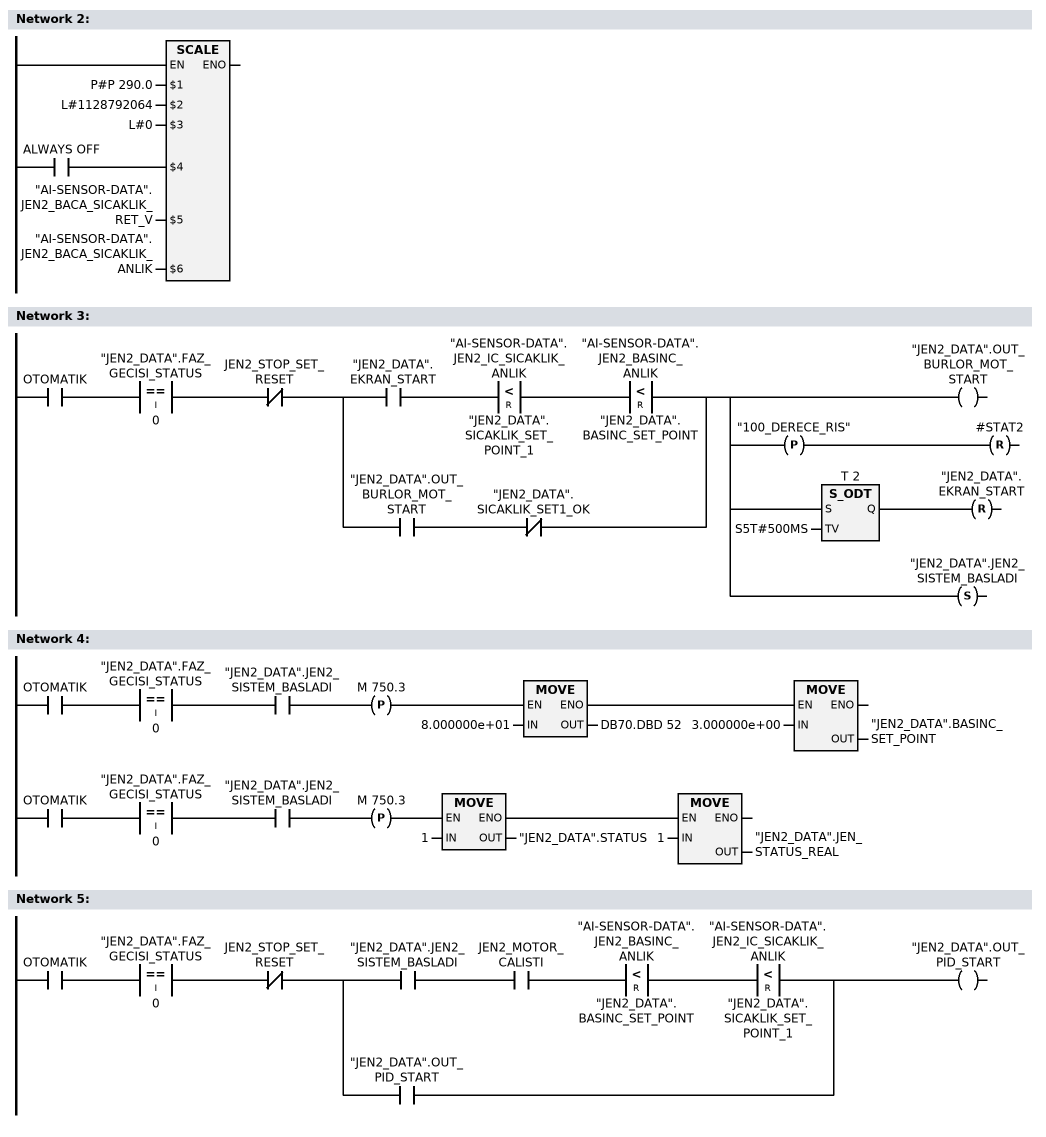
NETWORK
TITLE =
      A     "ALWAYS OFF";
      =     L 0.0;
      BLD   103;
      CALL  "SCALE" (
           $1                       := P#P 290.0,
           $2                       := L#1128792064,
           $3                       := L#0,
           $4                       := L 0.0,
           $5                       := "AI-SENSOR-DATA".JEN2_BACA_SICAKLIK_RET_V,
           $6                       := "AI-SENSOR-DATA".JEN2_BACA_SICAKLIK_ANLIK);
      NOP   0;
NETWORK
TITLE =
      A     "OTOMATIK";
      A(;
      L     "JEN2_DATA".FAZ_GECISI_STATUS;
      L     0;
      ==I;
      );
      AN    "JEN2_STOP_SET_RESET";
      A(;
      A     "JEN2_DATA".EKRAN_START;
      A(;
      L     "AI-SENSOR-DATA".JEN2_IC_SICAKLIK_ANLIK;
      L     "JEN2_DATA".SICAKLIK_SET_POINT_1;
      <R;
      );
      A(;
      L     "AI-SENSOR-DATA".JEN2_BASINC_ANLIK;
      L     "JEN2_DATA".BASINC_SET_POINT;
      <R;
      );
      O;
      A     "JEN2_DATA".OUT_BURLOR_MOT_START;
      AN    "JEN2_DATA".SICAKLIK_SET1_OK;
      );
      =     L 0.0;
      A     L 0.0;
      BLD   102;
      =     "JEN2_DATA".OUT_BURLOR_MOT_START;
      A     L 0.0;
      FP    "100_DERECE_RIS";
      R     #STAT2;
      A     L 0.0;
      L     S5T#500MS;
      SD    T 2;
      NOP   0;
      NOP   0;
      NOP   0;
      A     T 2;
      R     "JEN2_DATA".EKRAN_START;
      A     L 0.0;
      BLD   102;
      S     "JEN2_DATA".JEN2_SISTEM_BASLADI;
NETWORK
TITLE =
      A     "OTOMATIK";
      A(;
      L     "JEN2_DATA".FAZ_GECISI_STATUS;
      L     0;
      ==I;
      );
      A     "JEN2_DATA".JEN2_SISTEM_BASLADI;
      FP    M 750.3;
      =     L 0.0;
      A(;
      A     L 0.0;
      JNB   _002;
      L     8.000000e+01;
      T     DB70.DBD 52;
      SET;
      SAVE;
      CLR;
_002: A     BR;
      );
      JNB   _003;
      L     3.000000e+00;
      T     "JEN2_DATA".BASINC_SET_POINT;
_003: NOP   0;
      A(;
      A     L 0.0;
      JNB   _004;
      L     1;
      T     "JEN2_DATA".STATUS;
      SET;
      SAVE;
      CLR;
_004: A     BR;
      );
      JNB   _005;
      L     1;
      T     "JEN2_DATA".JEN_STATUS_REAL;
_005: NOP   0;
NETWORK
TITLE =
      A     "OTOMATIK";
      A(;
      L     "JEN2_DATA".FAZ_GECISI_STATUS;
      L     0;
      ==I;
      );
      AN    "JEN2_STOP_SET_RESET";
      A(;
      A     "JEN2_DATA".JEN2_SISTEM_BASLADI;
      A     "JEN2_MOTOR_CALISTI";
      A(;
      L     "AI-SENSOR-DATA".JEN2_BASINC_ANLIK;
      L     "JEN2_DATA".BASINC_SET_POINT;
      <R;
      );
      A(;
      L     "AI-SENSOR-DATA".JEN2_IC_SICAKLIK_ANLIK;
      L     "JEN2_DATA".SICAKLIK_SET_POINT_1;
      <R;
      );
      O     "JEN2_DATA".OUT_PID_START;
      );
      =     "JEN2_DATA".OUT_PID_START;
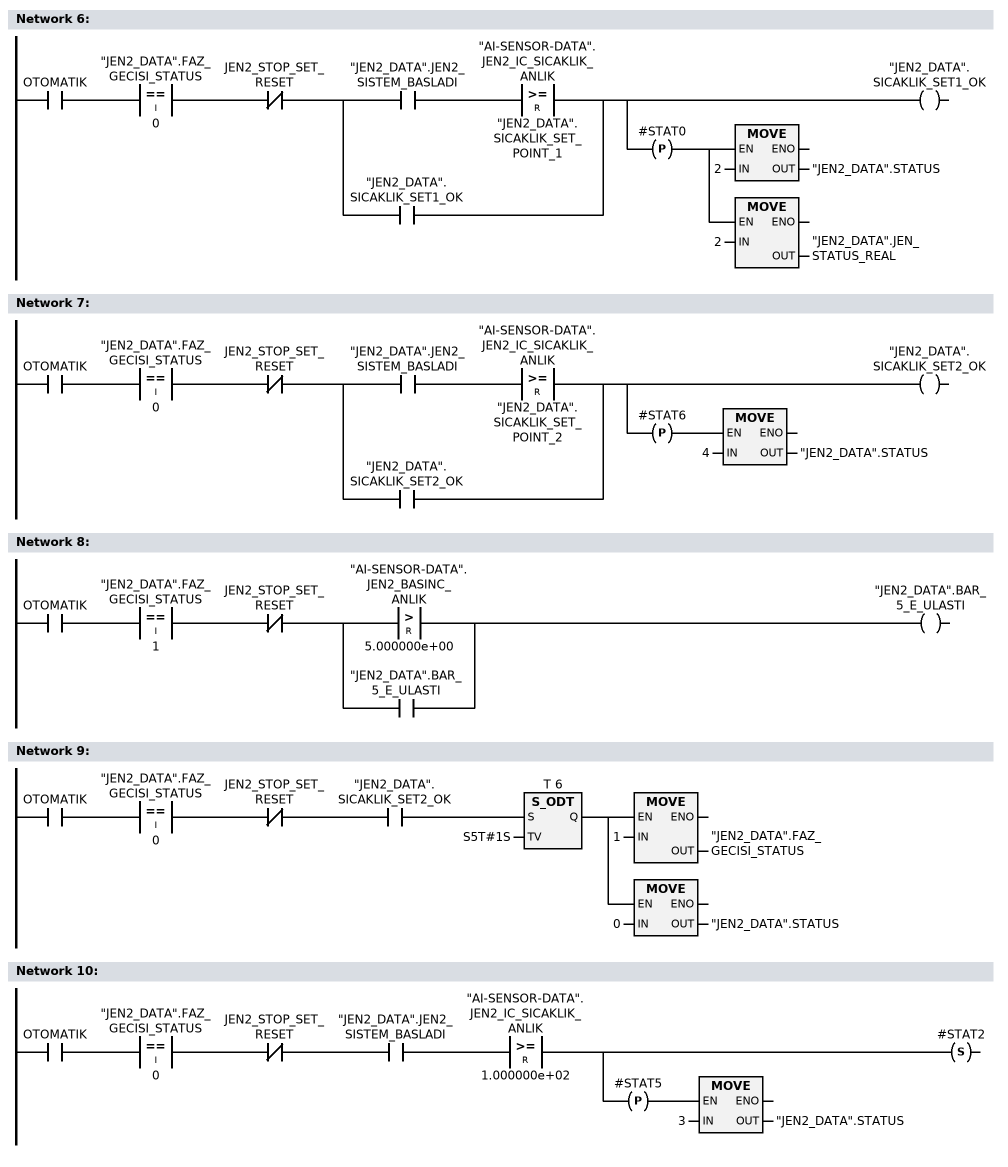
NETWORK
TITLE =
      A     "OTOMATIK";
      A(;
      L     "JEN2_DATA".FAZ_GECISI_STATUS;
      L     0;
      ==I;
      );
      AN    "JEN2_STOP_SET_RESET";
      A(;
      A     "JEN2_DATA".JEN2_SISTEM_BASLADI;
      A(;
      L     "AI-SENSOR-DATA".JEN2_IC_SICAKLIK_ANLIK;
      L     "JEN2_DATA".SICAKLIK_SET_POINT_1;
      >=R;
      );
      O     "JEN2_DATA".SICAKLIK_SET1_OK;
      );
      =     L 0.0;
      A     L 0.0;
      BLD   102;
      =     "JEN2_DATA".SICAKLIK_SET1_OK;
      A     L 0.0;
      FP    #STAT0;
      =     L 0.1;
      A     L 0.1;
      JNB   _006;
      L     2;
      T     "JEN2_DATA".STATUS;
_006: NOP   0;
      A     L 0.1;
      JNB   _007;
      L     2;
      T     "JEN2_DATA".JEN_STATUS_REAL;
_007: NOP   0;
NETWORK
TITLE =
      A     "OTOMATIK";
      A(;
      L     "JEN2_DATA".FAZ_GECISI_STATUS;
      L     0;
      ==I;
      );
      AN    "JEN2_STOP_SET_RESET";
      A(;
      A     "JEN2_DATA".JEN2_SISTEM_BASLADI;
      A(;
      L     "AI-SENSOR-DATA".JEN2_IC_SICAKLIK_ANLIK;
      L     "JEN2_DATA".SICAKLIK_SET_POINT_2;
      >=R;
      );
      O     "JEN2_DATA".SICAKLIK_SET2_OK;
      );
      =     L 0.0;
      A     L 0.0;
      BLD   102;
      =     "JEN2_DATA".SICAKLIK_SET2_OK;
      A     L 0.0;
      FP    #STAT6;
      JNB   _008;
      L     4;
      T     "JEN2_DATA".STATUS;
_008: NOP   0;
NETWORK
TITLE =
      A     "OTOMATIK";
      A(;
      L     "JEN2_DATA".FAZ_GECISI_STATUS;
      L     1;
      ==I;
      );
      AN    "JEN2_STOP_SET_RESET";
      A(;
      O(;
      L     "AI-SENSOR-DATA".JEN2_BASINC_ANLIK;
      L     5.000000e+00;
      >R;
      );
      O     "JEN2_DATA".BAR_5_E_ULASTI;
      );
      =     "JEN2_DATA".BAR_5_E_ULASTI;
NETWORK
TITLE =
      A     "OTOMATIK";
      A(;
      L     "JEN2_DATA".FAZ_GECISI_STATUS;
      L     0;
      ==I;
      );
      AN    "JEN2_STOP_SET_RESET";
      A     "JEN2_DATA".SICAKLIK_SET2_OK;
      L     S5T#1S;
      SD    T 6;
      NOP   0;
      NOP   0;
      NOP   0;
      A     T 6;
      =     L 0.0;
      A     L 0.0;
      JNB   _009;
      L     1;
      T     "JEN2_DATA".FAZ_GECISI_STATUS;
_009: NOP   0;
      A     L 0.0;
      JNB   _00a;
      L     0;
      T     "JEN2_DATA".STATUS;
_00a: NOP   0;
NETWORK
TITLE =
      A     "OTOMATIK";
      A(;
      L     "JEN2_DATA".FAZ_GECISI_STATUS;
      L     0;
      ==I;
      );
      AN    "JEN2_STOP_SET_RESET";
      A     "JEN2_DATA".JEN2_SISTEM_BASLADI;
      A(;
      L     "AI-SENSOR-DATA".JEN2_IC_SICAKLIK_ANLIK;
      L     1.000000e+02;
      >=R;
      );
      =     L 0.0;
      A     L 0.0;
      BLD   102;
      S     #STAT2;
      A     L 0.0;
      FP    #STAT5;
      JNB   _00b;
      L     3;
      T     "JEN2_DATA".STATUS;
_00b: NOP   0;
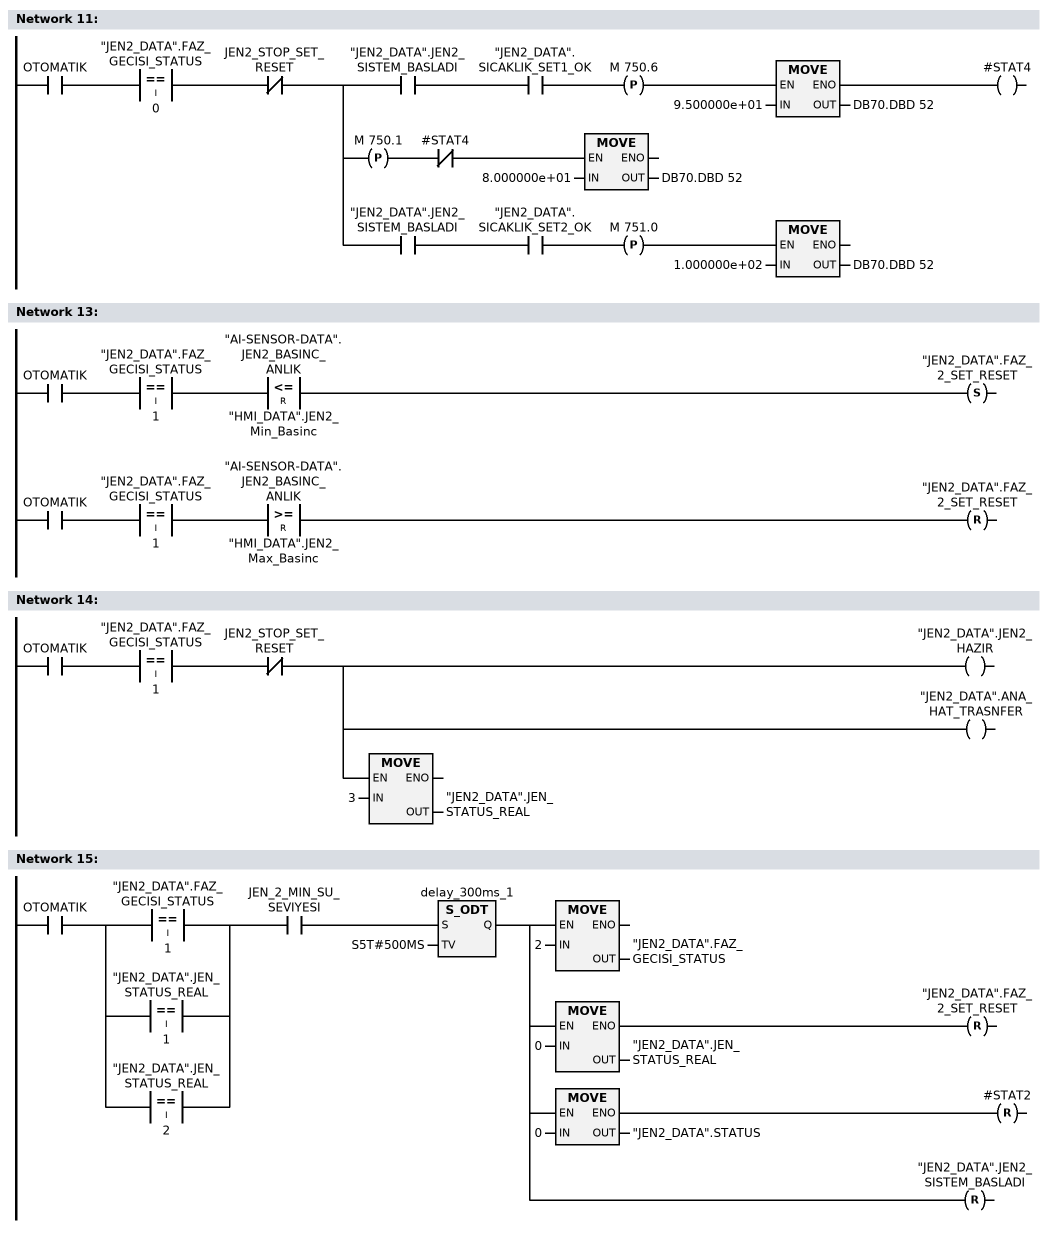
NETWORK
TITLE =
      A     "OTOMATIK";
      A(;
      L     "JEN2_DATA".FAZ_GECISI_STATUS;
      L     0;
      ==I;
      );
      AN    "JEN2_STOP_SET_RESET";
      =     L 0.0;
      A     L 0.0;
      A     "JEN2_DATA".JEN2_SISTEM_BASLADI;
      A     "JEN2_DATA".SICAKLIK_SET1_OK;
      FP    M 750.6;
      JNB   _00c;
      L     9.500000e+01;
      T     DB70.DBD 52;
      SET;
      SAVE;
      CLR;
_00c: A     BR;
      =     #STAT4;
      A     L 0.0;
      FP    M 750.1;
      AN    #STAT4;
      JNB   _00d;
      L     8.000000e+01;
      T     DB70.DBD 52;
_00d: NOP   0;
      A     L 0.0;
      A     "JEN2_DATA".JEN2_SISTEM_BASLADI;
      A     "JEN2_DATA".SICAKLIK_SET2_OK;
      FP    M 751.0;
      JNB   _00e;
      L     1.000000e+02;
      T     DB70.DBD 52;
_00e: NOP   0;
NETWORK
TITLE =
NETWORK
TITLE =
      A     "OTOMATIK";
      A(;
      L     "JEN2_DATA".FAZ_GECISI_STATUS;
      L     1;
      ==I;
      );
      A(;
      L     "AI-SENSOR-DATA".JEN2_BASINC_ANLIK;
      L     "HMI_DATA".JEN2_Min_Basinc;
      <=R;
      );
      S     "JEN2_DATA".FAZ_2_SET_RESET;
      A     "OTOMATIK";
      A(;
      L     "JEN2_DATA".FAZ_GECISI_STATUS;
      L     1;
      ==I;
      );
      A(;
      L     "AI-SENSOR-DATA".JEN2_BASINC_ANLIK;
      L     "HMI_DATA".JEN2_Max_Basinc;
      >=R;
      );
      R     "JEN2_DATA".FAZ_2_SET_RESET;
      NOP   0;
NETWORK
TITLE =
      A     "OTOMATIK";
      A(;
      L     "JEN2_DATA".FAZ_GECISI_STATUS;
      L     1;
      ==I;
      );
      AN    "JEN2_STOP_SET_RESET";
      =     L 0.0;
      A     L 0.0;
      BLD   102;
      =     "JEN2_DATA".JEN2_HAZIR;
      A     L 0.0;
      BLD   102;
      =     "JEN2_DATA".ANA_HAT_TRASNFER;
      A     L 0.0;
      JNB   _00f;
      L     3;
      T     "JEN2_DATA".JEN_STATUS_REAL;
_00f: NOP   0;
NETWORK
TITLE =
      A     "OTOMATIK";
      A(;
      O(;
      L     "JEN2_DATA".FAZ_GECISI_STATUS;
      L     1;
      ==I;
      );
      O(;
      L     "JEN2_DATA".JEN_STATUS_REAL;
      L     1;
      ==I;
      );
      O(;
      L     "JEN2_DATA".JEN_STATUS_REAL;
      L     2;
      ==I;
      );
      );
      A     "JEN_2_MIN_SU_SEVIYESI";
      L     S5T#500MS;
      SD    "delay_300ms_1";
      NOP   0;
      NOP   0;
      NOP   0;
      A     "delay_300ms_1";
      =     L 0.0;
      A     L 0.0;
      JNB   _010;
      L     2;
      T     "JEN2_DATA".FAZ_GECISI_STATUS;
_010: NOP   0;
      A     L 0.0;
      JNB   _011;
      L     0;
      T     "JEN2_DATA".JEN_STATUS_REAL;
      SET;
      SAVE;
      CLR;
_011: A     BR;
      R     "JEN2_DATA".FAZ_2_SET_RESET;
      A     L 0.0;
      JNB   _012;
      L     0;
      T     "JEN2_DATA".STATUS;
      SET;
      SAVE;
      CLR;
_012: A     BR;
      R     #STAT2;
      A     L 0.0;
      BLD   102;
      R     "JEN2_DATA".JEN2_SISTEM_BASLADI;
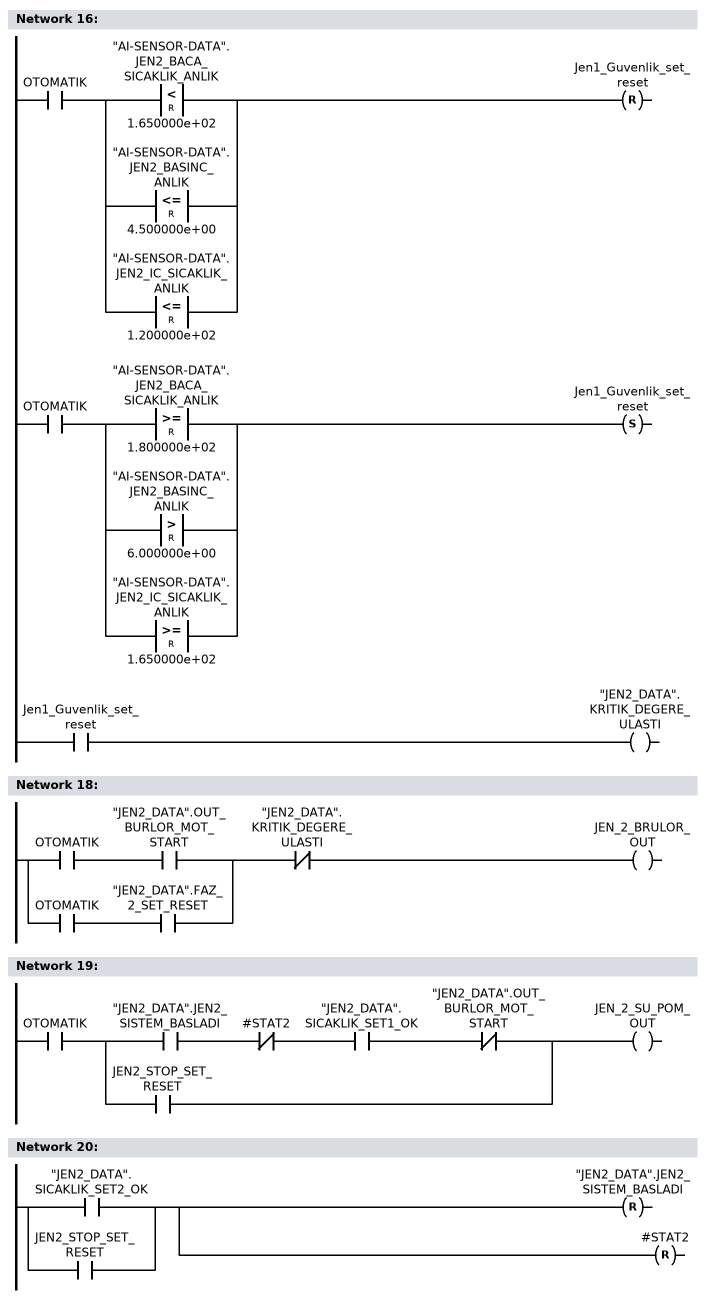
NETWORK
TITLE =
      A     "OTOMATIK";
      A(;
      O(;
      L     "AI-SENSOR-DATA".JEN2_BACA_SICAKLIK_ANLIK;
      L     1.650000e+02;
      <R;
      );
      O(;
      L     "AI-SENSOR-DATA".JEN2_BASINC_ANLIK;
      L     4.500000e+00;
      <=R;
      );
      O(;
      L     "AI-SENSOR-DATA".JEN2_IC_SICAKLIK_ANLIK;
      L     1.200000e+02;
      <=R;
      );
      );
      R     "Jen1_Guvenlik_set_reset";
      A     "OTOMATIK";
      A(;
      O(;
      L     "AI-SENSOR-DATA".JEN2_BACA_SICAKLIK_ANLIK;
      L     1.800000e+02;
      >=R;
      );
      O(;
      L     "AI-SENSOR-DATA".JEN2_BASINC_ANLIK;
      L     6.000000e+00;
      >R;
      );
      O(;
      L     "AI-SENSOR-DATA".JEN2_IC_SICAKLIK_ANLIK;
      L     1.650000e+02;
      >=R;
      );
      );
      S     "Jen1_Guvenlik_set_reset";
      A     "Jen1_Guvenlik_set_reset";
      =     "JEN2_DATA".KRITIK_DEGERE_ULASTI;
NETWORK
TITLE =
NETWORK
TITLE =
      A(;
      A     "OTOMATIK";
      A     "JEN2_DATA".OUT_BURLOR_MOT_START;
      O;
      A     "OTOMATIK";
      A     "JEN2_DATA".FAZ_2_SET_RESET;
      );
      AN    "JEN2_DATA".KRITIK_DEGERE_ULASTI;
      =     "JEN_2_BRULOR_OUT";
NETWORK
TITLE =
      A     "OTOMATIK";
      A(;
      A     "JEN2_DATA".JEN2_SISTEM_BASLADI;
      AN    #STAT2;
      A     "JEN2_DATA".SICAKLIK_SET1_OK;
      AN    "JEN2_DATA".OUT_BURLOR_MOT_START;
      O     "JEN2_STOP_SET_RESET";
      );
      =     "JEN_2_SU_POM_OUT";
NETWORK
TITLE =
      O     "JEN2_DATA".SICAKLIK_SET2_OK;
      O     "JEN2_STOP_SET_RESET";
      R     "JEN2_DATA".JEN2_SISTEM_BASLADI;
      R     #STAT2;
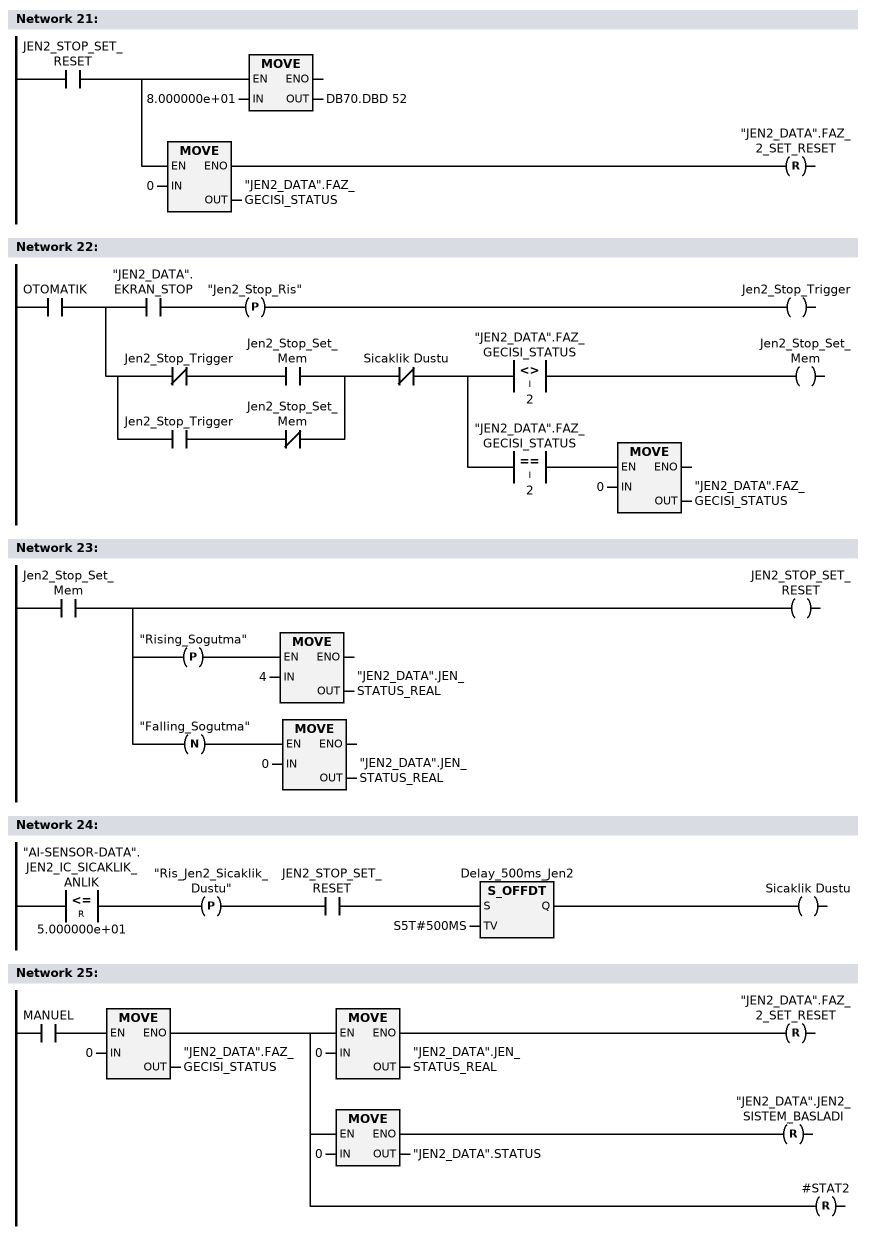
NETWORK
TITLE =
      A     "JEN2_STOP_SET_RESET";
      =     L 0.0;
      A     L 0.0;
      JNB   _013;
      L     8.000000e+01;
      T     DB70.DBD 52;
_013: NOP   0;
      A     L 0.0;
      JNB   _014;
      L     0;
      T     "JEN2_DATA".FAZ_GECISI_STATUS;
      SET;
      SAVE;
      CLR;
_014: A     BR;
      R     "JEN2_DATA".FAZ_2_SET_RESET;
NETWORK
TITLE =
      A     "OTOMATIK";
      =     L 0.0;
      A     L 0.0;
      A     "JEN2_DATA".EKRAN_STOP;
      FP    "Jen2_Stop_Ris";
      =     "Jen2_Stop_Trigger";
      A     L 0.0;
      A(;
      AN    "Jen2_Stop_Trigger";
      A     "Jen2_Stop_Set_Mem";
      O;
      A     "Jen2_Stop_Trigger";
      AN    "Jen2_Stop_Set_Mem";
      );
      AN    "Sicaklik Dustu";
      =     L 0.1;
      A     L 0.1;
      A(;
      L     "JEN2_DATA".FAZ_GECISI_STATUS;
      L     2;
      <>I;
      );
      =     "Jen2_Stop_Set_Mem";
      A     L 0.1;
      A(;
      L     "JEN2_DATA".FAZ_GECISI_STATUS;
      L     2;
      ==I;
      );
      JNB   _015;
      L     0;
      T     "JEN2_DATA".FAZ_GECISI_STATUS;
_015: NOP   0;
NETWORK
TITLE =
      A     "Jen2_Stop_Set_Mem";
      =     L 0.0;
      A     L 0.0;
      BLD   102;
      =     "JEN2_STOP_SET_RESET";
      A     L 0.0;
      FP    "Rising_Sogutma";
      JNB   _016;
      L     4;
      T     "JEN2_DATA".JEN_STATUS_REAL;
_016: NOP   0;
      A     L 0.0;
      FN    "Falling_Sogutma";
      JNB   _017;
      L     0;
      T     "JEN2_DATA".JEN_STATUS_REAL;
_017: NOP   0;
NETWORK
TITLE =
      A(;
      L     "AI-SENSOR-DATA".JEN2_IC_SICAKLIK_ANLIK;
      L     5.000000e+01;
      <=R;
      );
      FP    "Ris_Jen2_Sicaklik_Dustu";
      A     "JEN2_STOP_SET_RESET";
      L     S5T#500MS;
      SF    "Delay_500ms_Jen2";
      NOP   0;
      NOP   0;
      NOP   0;
      A     "Delay_500ms_Jen2";
      =     "Sicaklik Dustu";
NETWORK
TITLE =
      A     "MANUEL";
      JNB   _018;
      L     0;
      T     "JEN2_DATA".FAZ_GECISI_STATUS;
      SET;
      SAVE;
      CLR;
_018: A     BR;
      =     L 0.0;
      A     L 0.0;
      JNB   _019;
      L     0;
      T     "JEN2_DATA".JEN_STATUS_REAL;
      SET;
      SAVE;
      CLR;
_019: A     BR;
      R     "JEN2_DATA".FAZ_2_SET_RESET;
      A     L 0.0;
      JNB   _01a;
      L     0;
      T     "JEN2_DATA".STATUS;
      SET;
      SAVE;
      CLR;
_01a: A     BR;
      R     "JEN2_DATA".JEN2_SISTEM_BASLADI;
      A     L 0.0;
      BLD   102;
      R     #STAT2;
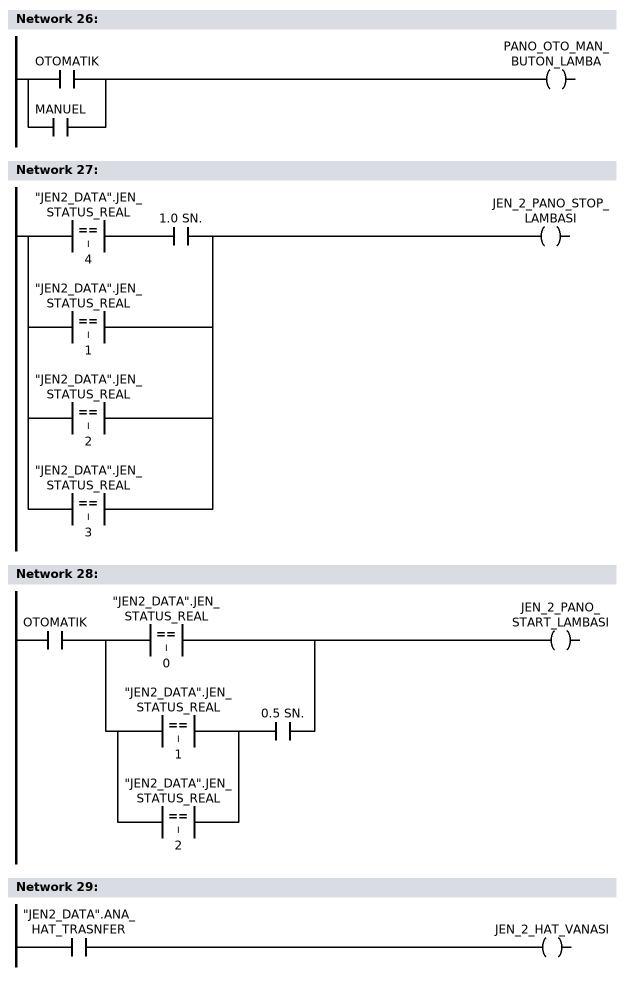
NETWORK
TITLE =
      O     "OTOMATIK";
      O     "MANUEL";
      =     "PANO_OTO_MAN_BUTON_LAMBA";
NETWORK
TITLE =
      A(;
      L     "JEN2_DATA".JEN_STATUS_REAL;
      L     4;
      ==I;
      );
      A     "1.0 SN.";
      O(;
      L     "JEN2_DATA".JEN_STATUS_REAL;
      L     1;
      ==I;
      );
      O(;
      L     "JEN2_DATA".JEN_STATUS_REAL;
      L     2;
      ==I;
      );
      O(;
      L     "JEN2_DATA".JEN_STATUS_REAL;
      L     3;
      ==I;
      );
      =     "JEN_2_PANO_STOP_LAMBASI";
NETWORK
TITLE =
      A     "OTOMATIK";
      A(;
      O(;
      L     "JEN2_DATA".JEN_STATUS_REAL;
      L     0;
      ==I;
      );
      O;
      A(;
      O(;
      L     "JEN2_DATA".JEN_STATUS_REAL;
      L     1;
      ==I;
      );
      O(;
      L     "JEN2_DATA".JEN_STATUS_REAL;
      L     2;
      ==I;
      );
      );
      A     "0.5 SN.";
      );
      =     "JEN_2_PANO_START_LAMBASI";
NETWORK
TITLE =
      A     "JEN2_DATA".ANA_HAT_TRASNFER;
      =     "JEN_2_HAT_VANASI";
END_FUNCTION_BLOCK

FUNCTION "TIME_UNSCALE" : VOID	// FC 1
VERSION : 0.0
BEGIN
// body was compiled from an SCL source; compiled code not shown
END_FUNCTION

FUNCTION "O.Vana_AciklikHesaplama" : VOID	// FC 2
VERSION : 0.1
VAR_INPUT
  IlkAciklikDegeri : REAL ;
  KademeliAcikDegeri : REAL ;
END_VAR
VAR_OUTPUT
  oKademe_1 : REAL ;
  oKademe_2 : REAL ;
  oKademe_3 : REAL ;
  oKademe_4 : REAL ;
  oKademe_5 : REAL ;
  oKademe_6 : REAL ;
  oKademe_7 : REAL ;
END_VAR
VAR_TEMP
  tKademe : STRUCT
   Iki : REAL ;
   Uc : REAL ;
   Dort : REAL ;
   Bes : REAL ;
   Alti : REAL ;
   Yedi : REAL ;
  END_STRUCT ;
  tCheck_Kademe5 : BOOL ;
  tCheck_Kademe6 : BOOL ;
  tCheck_Kademe7 : BOOL ;
END_VAR
BEGIN
NETWORK
TITLE =
//------------------------
// kademe 1
      L     #IlkAciklikDegeri;
      T     #oKademe_1;
//------------------------
// kademe 2
      L     #IlkAciklikDegeri;
      L     #KademeliAcikDegeri;
      +R;
      T     #tKademe.Iki;
      L     #tKademe.Iki;
      T     #oKademe_2;
//-----------------------
// kademe 3
      L     #KademeliAcikDegeri;
      L     #tKademe.Iki;
      +R;
      T     #tKademe.Uc;
      L     #tKademe.Uc;
      T     #oKademe_3;
//-----------------------
// kademe 4
      L     #KademeliAcikDegeri;
      L     #tKademe.Uc;
      +R;
      T     #tKademe.Dort;
      L     #tKademe.Dort;
      T     #oKademe_4;
//-----------------------
// kademe 5
      L     #KademeliAcikDegeri;
      L     #tKademe.Dort;
      +R;
      T     #tKademe.Bes;
      L     #tKademe.Bes;
      L     6.000000e+01;
      >R;
      =     #tCheck_Kademe5;
      A     #tCheck_Kademe5;
      JNB   j005;
      L     6.000000e+01;
      T     #tKademe.Bes;
j005: NOP   0;
      L     #tKademe.Bes;
      T     #oKademe_5;
//-----------------------
// kademe 6
      L     #KademeliAcikDegeri;
      L     #tKademe.Bes;
      +R;
      T     #tKademe.Alti;
      L     #tKademe.Alti;
      L     6.000000e+01;
      >R;
      =     #tCheck_Kademe6;
      A     #tCheck_Kademe6;
      JNB   j006;
      L     6.000000e+01;
      T     #tKademe.Alti;
j006: NOP   0;
      L     #tKademe.Alti;
      T     #oKademe_6;
//-----------------------
// kademe 7
      L     #KademeliAcikDegeri;
      L     #tKademe.Alti;
      +R;
      T     #tKademe.Yedi;
      L     #tKademe.Yedi;
      L     6.000000e+01;
      >R;
      =     #tCheck_Kademe7;
      A     #tCheck_Kademe7;
      JNB   j007;
      L     6.000000e+01;
      T     #tKademe.Yedi;
j007: NOP   0;
      L     #tKademe.Yedi;
      T     #oKademe_7;
NETWORK
TITLE =
END_FUNCTION

FUNCTION "Int_To_S5Time" : VOID	// FC 10
VERSION : 0.0
VAR_INPUT
  Saat : INT ;
  Dakika : INT ;
END_VAR
VAR_OUTPUT
  HesaplananSure_S5TIME : S5TIME ;
END_VAR
VAR_TEMP
  tSaat_Dint : DINT ;
  tHesaplananSaat : DINT ;
  tDakika_Dint : DINT ;
  tHesaplananDakika : DINT ;
  tHesaplnananSure_Dint : DINT ;
  tHesaplananSure_Time : TIME ;
END_VAR
BEGIN
// body was compiled from an SCL source; compiled code not shown
END_FUNCTION

FUNCTION "Int_To_Second" : VOID	// FC 11
VERSION : 0.0
VAR_INPUT
  Saniye : INT ;
END_VAR
VAR_OUTPUT
  HesaplananSure_S5TIME : S5TIME ;
END_VAR
VAR_TEMP
  tSaniye_Dint : DINT ;
  tHesaplananSaniye : DINT ;
  tHesaplnananSure_Dint : DINT ;
  tHesaplananSure_Time : TIME ;
END_VAR
BEGIN
// body was compiled from an SCL source; compiled code not shown
END_FUNCTION

// FC 33: know-how protected block, not included

// FC 40: know-how protected block, not included

// FC 105: know-how protected block, not included

// FC 106: know-how protected block, not included

DATA_BLOCK "AI-SENSOR-DATA"	// DB 1
VERSION : 0.1
  STRUCT
   JEN1_BASINC_ANLIK : REAL ;
   JEN2_BASINC_ANLIK : REAL ;
   JEN1_BASINC_RET_VAL : WORD ;
   JEN2_BASINC_RET_VAL : WORD ;
   JEN1_IC_SICAKLIK_ANLIK : REAL ;
   JEN2_IC_SICAKLIK_ANLIK : REAL ;
   JEN1_IC_SICAKLIK_RET_VAL : WORD ;
   JEN2_IC_SICAKLIK_RET_VAL : WORD ;
   JEN1_BACA_SICAKLIK_ANLIK : REAL ;
   JEN2_BACA_SICAKLIK_ANLIK : REAL ;
   JEN1_BACA_SICAKLIK_RET_V : WORD ;
   JEN2_BACA_SICAKLIK_RET_V : WORD ;
   HAT_BASINCI_RET_V : WORD ;
   HAT_BASINCI_ANLIK : REAL ;
   HAVA_BASINCI_RET_V : WORD ;
   HAVA_BASINCI_ANLIK : REAL ;
   HAT_BASINCI_YETERLI : BOOL ;
  END_STRUCT ;	
BEGIN
   JEN1_BASINC_ANLIK := 4.452402e+00;
   JEN2_BASINC_RET_VAL := W#16#8;
   JEN1_IC_SICAKLIK_ANLIK := 1.514829e+02;
   JEN2_IC_SICAKLIK_ANLIK := 2.052228e+01;
   JEN1_BACA_SICAKLIK_ANLIK := 5.423901e+01;
   JEN2_BACA_SICAKLIK_ANLIK := 9.780092e+00;
   HAT_BASINCI_ANLIK := 4.622757e+00;
   HAVA_BASINCI_ANLIK := 4.994936e+00;
   HAT_BASINCI_YETERLI := TRUE;
END_DATA_BLOCK

DATA_BLOCK "ORTAK_DATA"	// DB 2
VERSION : 0.1
  STRUCT
   JEN_EMNIYET_BASINCI : REAL ;
   JEN_EMNIYET_SICAKLIGI : REAL ;
   OTO_EMNIYET_BASINCI : REAL ;
   OTO_EMNIYET_SICAKLIGI : REAL ;
   OTO_ISLEM_BITTI_VANA_AC : BOOL ;
   OTO_JEN_DURDU : REAL ;
  END_STRUCT ;	
BEGIN
END_DATA_BLOCK

DATA_BLOCK "TIME_OTO_1_DB"	// DB 5
AUTHOR : SIMATIC
FAMILY : IEC_TC
VERSION : 0.0
"TON"
BEGIN
END_DATA_BLOCK

DATA_BLOCK "TIME_OTO_2_DB"	// DB 6
AUTHOR : SIMATIC
FAMILY : IEC_TC
VERSION : 0.0
"TON"
BEGIN
END_DATA_BLOCK

DATA_BLOCK "TIME_OTO_1_PROSES_DB"	// DB 7
AUTHOR : SIMATIC
FAMILY : IEC_TC
VERSION : 0.0
"TON"
BEGIN
END_DATA_BLOCK

DATA_BLOCK "TIME_OTO_2_PROSES_DB"	// DB 8
AUTHOR : SIMATIC
FAMILY : IEC_TC
VERSION : 0.0
"TON"
BEGIN
END_DATA_BLOCK

DATA_BLOCK DB 9
AUTHOR : SIMATIC
FAMILY : IEC_TC
VERSION : 0.0
"TON"
BEGIN
END_DATA_BLOCK

DATA_BLOCK DB 10
AUTHOR : SIMATIC
FAMILY : IEC_TC
VERSION : 0.0
"TON"
BEGIN
END_DATA_BLOCK

DATA_BLOCK "SURELER_DB"	// DB 14
VERSION : 0.0
"SURELER"
BEGIN
END_DATA_BLOCK

DATA_BLOCK "SAFETY_DB"	// DB 15
VERSION : 0.0
"SAFETY"
BEGIN
END_DATA_BLOCK

DATA_BLOCK "KAZAN1_DATA"	// DB 17
VERSION : 0.1
  STRUCT
   IN_STATUS : INT ;
   IN_JEN_OK : BOOL ;
   IN_DIGER_KAZ_TRANS_HAZIR : BOOL ;
   IN_PISIM_SURESI : S5TIME ;
   IN_SCALE_BASINC_PER : INT ;
   IN_SET_BASINC : REAL ;
   IN_DIGER_KAZAN_BASINCI : REAL ;
   O_PID_MAN_ON : BOOL ;
   O_PID_MAN : REAL ;
   O_TRANSFER_YAPILIYOR : BOOL ;
   O_SCALE_BASINC_RET_VAL : WORD ;
   O_SCALE_BASINC_OUT : REAL ;
   O_TRANSFERE_HAZIR : BOOL ;
   O_SCALE_SICAKLIK_RET_VAL : WORD ;
   O_SCALE_SICAKLIK_OUT : REAL ;
   IN_SCALE_SICAKLIK_PER : INT ;
   O_KAZAN_BOSALTIMDA : BOOL ;
   IN_DIGER_KAZ_BOSALTIMDA : BOOL ;
   IN_DIGER_KAZ_TRANSFERDE : BOOL ;
   O_PISIM_BASLADI : BOOL ;
   PISIM_GECEN_SURE_TIME : TIME ;
   PISIM_GECEN_SURE_DINT : DINT ;
   PROSES_SURESI_TIME : TIME ;
   PROSES_SURESI_DINT : DINT ;
   BEKLEME_SURESI_TIME : TIME ;
   BEKLEME_SURESI_DINT : DINT ;
  END_STRUCT ;	
BEGIN
   IN_JEN_OK := TRUE;
   IN_PISIM_SURESI := S5T#21M;
   IN_SCALE_BASINC_PER := 3;
   IN_SET_BASINC := 4.500000e+00;
   IN_DIGER_KAZAN_BASINCI := 3.616898e-03;
   O_SCALE_BASINC_OUT := 3.978588e-03;
   O_SCALE_SICAKLIK_OUT := 5.775463e+01;
   IN_SCALE_SICAKLIK_PER := 7969;
   PISIM_GECEN_SURE_DINT := L#1260;
END_DATA_BLOCK

DATA_BLOCK "KAZAN2_DATA"	// DB 18
VERSION : 0.1
  STRUCT
   IN_STATUS : INT ;
   IN_JEN_OK : BOOL ;
   IN_DIGER_KAZ_TRANS_HAZIR : BOOL ;
   IN_PISIM_SURESI : S5TIME ;
   IN_SCALE_BASINC_PER : INT ;
   IN_SET_BASINC : REAL ;
   IN_DIGER_KAZAN_BASINCI : REAL ;
   O_PID_MAN_ON : BOOL ;
   O_PID_MAN : REAL ;
   O_TRANSFER_YAPILIYOR : BOOL ;
   O_SCALE_BASINC_RET_VAL : WORD ;
   O_SCALE_BASINC_OUT : REAL ;
   O_TRANSFERE_HAZIR : BOOL ;
   O_SCALE_SICAKLIK_RET_VAL : WORD ;
   O_SCALE_SICAKLIK_OUT : REAL ;
   IN_SCALE_SICAKLIK_PER : INT ;
   O_KAZAN_BOSALTIMDA : BOOL ;
   IN_DIGER_KAZ_BOSALTIMDA : BOOL ;
   IN_DIGER_KAZ_TRANSFERDE : BOOL ;
   O_PISIM_BASLADI : BOOL ;
   PISIM_GECEN_SURE_TIME : TIME ;
   PISIM_GECEN_SURE_DINT : DINT ;
   PROSES_SURESI_TIM : TIME ;
   PROSES_SURESI_DINT : DINT ;
   BEKLEME_SURESI_TIME : TIME ;
   BEKLEME_SURESI_DINT : DINT ;
  END_STRUCT ;	
BEGIN
   IN_JEN_OK := TRUE;
   IN_PISIM_SURESI := S5T#21M;
   IN_SCALE_BASINC_PER := -23;
   IN_SET_BASINC := 4.500000e+00;
   IN_DIGER_KAZAN_BASINCI := 2.857350e-02;
   O_SCALE_BASINC_OUT := 4.701968e-03;
   O_SCALE_SICAKLIK_OUT := 1.045356e+02;
   IN_SCALE_SICAKLIK_PER := 14476;
   PISIM_GECEN_SURE_DINT := L#1260;
END_DATA_BLOCK

DATA_BLOCK "JEN1_DATA"	// DB 19
VERSION : 0.1
  STRUCT
   BASINC_SET_POINT : REAL ;
   STATUS : INT ;
   SICAKLIK_SET_POINT_1 : REAL ;
   SICAKLIK_SET_POINT_2 : REAL ;
   SISTEM_BASLADI : BOOL ;
   EKRAN_START : BOOL ;
   EKRAN_STOP : BOOL ;
   OUT_BURLOR_MOT_START : BOOL ;
   SICAKLIK_SET1_OK : BOOL ;
   SICAKLIK_SET2_OK : BOOL ;
   OUT_PID_START : BOOL ;
   FAZ_GECISI_STATUS : INT ;
   FAZ_2_SET_RESET : BOOL ;
   BAR_5_E_ULASTI : BOOL ;
   JEN1_HAZIR : BOOL ;
   ANA_HAT_TRASFER_HAZIR : BOOL ;
   JEN_STATUS_REAL : INT ;
   STOP_SET_RESET : BOOL ;
   CALISMA_SURESI_TIME : TIME ;
   CALISMA_SURESI_DINT : DINT ;
   KRITIK_DEGERLERE_ULASTI : BOOL ;
   CALISMA_SURESI_EKRAN : DINT ;
   SET2_DEGERINE_ULASMADI : BOOL ;
  END_STRUCT ;	
BEGIN
   BASINC_SET_POINT := 3.000000e+00;
   SICAKLIK_SET_POINT_1 := 1.050000e+02;
   SICAKLIK_SET_POINT_2 := 1.300000e+02;
   FAZ_GECISI_STATUS := 1;
   FAZ_2_SET_RESET := TRUE;
   BAR_5_E_ULASTI := TRUE;
   JEN1_HAZIR := TRUE;
   ANA_HAT_TRASFER_HAZIR := TRUE;
   JEN_STATUS_REAL := 3;
   CALISMA_SURESI_DINT := L#32124;
END_DATA_BLOCK

DATA_BLOCK "JEN2_DATA"	// DB 20
VERSION : 0.1
  STRUCT
   BASINC_SET_POINT : REAL ;
   STATUS : INT ;
   SICAKLIK_SET_POINT_1 : REAL ;
   SICAKLIK_SET_POINT_2 : REAL ;
   JEN2_SISTEM_BASLADI : BOOL ;
   EKRAN_START : BOOL ;
   EKRAN_STOP : BOOL ;
   OUT_BURLOR_MOT_START : BOOL ;
   SICAKLIK_SET1_OK : BOOL ;
   SICAKLIK_SET2_OK : BOOL ;
   OUT_PID_START : BOOL ;
   FAZ_GECISI_STATUS : INT ;
   FAZ_2_SET_RESET : BOOL ;
   BAR_5_E_ULASTI : BOOL ;
   JEN2_HAZIR : BOOL ;
   ANA_HAT_TRASNFER : BOOL ;
   JEN_STATUS_REAL : INT ;
   STOP_SET_RESET : BOOL ;
   CALISMA_SURESI_TIME : TIME ;
   CALISMA_SURESI_DINT : DINT ;
   KRITIK_DEGERE_ULASTI : BOOL ;
   CALISMA_SURESI_EKRAN : DINT ;
  END_STRUCT ;	
BEGIN
   BASINC_SET_POINT := 3.000000e+00;
   SICAKLIK_SET_POINT_1 := 5.500000e+01;
   SICAKLIK_SET_POINT_2 := 1.100000e+02;
END_DATA_BLOCK

DATA_BLOCK "JEN1_PID_DATA"	// DB 21
VERSION : 0.1
  STRUCT
   TCONT_C_LMN : REAL ;
   TCONT_C_LMN_PER : INT ;
  END_STRUCT ;	
BEGIN
END_DATA_BLOCK

DATA_BLOCK "JEN2_PID_DATA"	// DB 22
VERSION : 0.1
  STRUCT
   TCONT_C_LMN : REAL ;
   TCONT_C_LMN_PER : INT ;
  END_STRUCT ;	
BEGIN
   TCONT_C_LMN_PER := 11059;
END_DATA_BLOCK

DATA_BLOCK "KAZAN1_PID_DATA"	// DB 23
VERSION : 0.1
  STRUCT
   TCONT_LMN_PER : INT ;
   TCONT_LMN : REAL ;
  END_STRUCT ;	
BEGIN
END_DATA_BLOCK

DATA_BLOCK "KAZAN2_PID_DATA"	// DB 24
VERSION : 0.1
  STRUCT
   TCONT_LMN_PER : INT ;
   TCONT_LMN : REAL ;
  END_STRUCT ;	
BEGIN
END_DATA_BLOCK

DATA_BLOCK DB 50
AUTHOR : SIMATIC
FAMILY : ICONT
VERSION : 0.0
"CONT_C"
BEGIN
END_DATA_BLOCK

DATA_BLOCK "JEN2_KONTROL_BLOGU_DB"	// DB 51
VERSION : 0.0
"JEN2_PID_KONTROL"
BEGIN
END_DATA_BLOCK

DATA_BLOCK DB 52
VERSION : 0.0
"JEN1_PID_KONTROL"
BEGIN
END_DATA_BLOCK

DATA_BLOCK "JEN_1_PID_DB"	// DB 69
AUTHOR : SIMATIC
FAMILY : CONTROL
VERSION : 0.0
"TCONT_CP"
BEGIN
END_DATA_BLOCK

DATA_BLOCK "JEN_2_PID_DB"	// DB 70
AUTHOR : SIMATIC
FAMILY : CONTROL
VERSION : 0.0
"TCONT_CP"
BEGIN
END_DATA_BLOCK

DATA_BLOCK "OTOKLAV_1_DB"	// DB 94
VERSION : 0.0
"KAZAN_1_KONTROL"
BEGIN
END_DATA_BLOCK

DATA_BLOCK "OTOKLAV_2_DB"	// DB 95
VERSION : 0.0
"KAZAN_2_KONTROL"
BEGIN
END_DATA_BLOCK

DATA_BLOCK "FB98_DB"	// DB 98
VERSION : 0.0
"JEN1_KONTROL_BLOGU"
BEGIN
END_DATA_BLOCK

DATA_BLOCK "FB99_DB"	// DB 99
VERSION : 0.0
"JEN2_KONTROL_BLOGU"
BEGIN
END_DATA_BLOCK

DATA_BLOCK "HMI_DATA"	// DB 100
VERSION : 0.1
  STRUCT
   JEN1_Min_Basinc : REAL  := 5.000000e+000;	//Jenerator 1 min otomatik sekans basinci
   JEN1_Max_Basinc : REAL  := 5.500000e+000;	//Jenerator 1 max otomatik sekans basinci
   JEN2_Min_Basinc : REAL  := 5.000000e+000;	//Jenerator 2 min otomatik sekans basinci
   JEN2_Max_Basinc : REAL  := 5.500000e+000;	//Jenerator 2 max otomatik sekans basinci
   OTOKLAV_First_Oran : REAL  := 2.000000e+001;	//Otoklav oransal vana otomatik sekans ilk acilis orani
   OTOKLAV_Kademeli_Artis : REAL  := 5.000000e+000;	//Otoklav oransal vana kademeli artis katsayisi
   Otoklav_1_TimeData : STRUCT 	//Otoklav 1 hmi süre bilgisi
    Hours : INT ;	//Istenen calisma saati
    Minutes : INT  := 30;	//Istenen calisma dakikasi
    Second : INT ;	//Istenen calisma saniyesi
   END_STRUCT ;
   Otoklav_2_TimeData : STRUCT 	//Otoklav 2 hmi süre bilgisi
    Hours : INT ;	//Istenen calisma saati
    Minutes : INT  := 30;	//Istenen calisma dakikasi
    Second : INT ;	//Istenen calisma saniyesi
   END_STRUCT ;
   O_VanaAciklikOrani : REAL  := 2.500000e+001;	//Oransal vana aciklik orani
   O_VanaKademeSayisi : REAL  := 5.000000e+000;	//Oransal vana kademeli artis katsayisi
   Otoklav1_Bos_Vanasi : STRUCT 	//Otoklav 1 Bosaltim Vanasi
    Vana_Acilma_Sayisi : INT  := 3;
    Periyod_Bekleme_Suresi : INT  := 120;	//Saniye bazinda
    Acik_Kalma_Suresi : INT  := 10;	//Saniye bazinda
   END_STRUCT ;
   Otoklav2_Bos_Vanasi : STRUCT 	//Otoklav 2 Bosaltim Vanasi
    Vana_Acilma_Sayisi : INT  := 3;
    Periyod_Bekleme_Suresi : INT  := 120;	//Saniye bazinda
    Acik_Kalma_Suresi : INT  := 10;	//Saniye bazinda
   END_STRUCT ;
   BosIsl_BosVana_Basinc : REAL  := 5.000000e-001;	//Bosaltim islemi sirasinda bosaltim vanas kapanma ve emniyet valf acilma basinci
  END_STRUCT ;	
BEGIN
   JEN1_Min_Basinc := 5.000000e+00;
   JEN1_Max_Basinc := 5.500000e+00;
   JEN2_Min_Basinc := 5.000000e+00;
   JEN2_Max_Basinc := 5.500000e+00;
   Otoklav_1_TimeData.Minutes := 30;
   Otoklav_2_TimeData.Minutes := 30;
   Otoklav1_Bos_Vanasi.Vana_Acilma_Sayisi := 3;
   Otoklav1_Bos_Vanasi.Periyod_Bekleme_Suresi := 120;
   Otoklav1_Bos_Vanasi.Acik_Kalma_Suresi := 10;
   Otoklav2_Bos_Vanasi.Vana_Acilma_Sayisi := 3;
   Otoklav2_Bos_Vanasi.Periyod_Bekleme_Suresi := 120;
   Otoklav2_Bos_Vanasi.Acik_Kalma_Suresi := 10;
   BosIsl_BosVana_Basinc := 5.000000e-01;
END_DATA_BLOCK

DATA_BLOCK DB 120
VERSION : 0.0
"KAZAN_ORTAK"
BEGIN
END_DATA_BLOCK

DATA_BLOCK "KAZAN_1_PID_DB"	// DB 130
AUTHOR : SIMATIC
FAMILY : CONTROL
VERSION : 0.0
"TCONT_CP"
BEGIN
END_DATA_BLOCK

DATA_BLOCK DB 131
VERSION : 0.0
"KAZAN_1_PID_KONTROL"
BEGIN
END_DATA_BLOCK

DATA_BLOCK DB 132
VERSION : 0.0
"KAZAN_2_PID_KONTROL"
BEGIN
END_DATA_BLOCK

DATA_BLOCK DB 230
VERSION : 0.0
"KAZAN_ORTAK"
BEGIN
END_DATA_BLOCK

DATA_BLOCK "KAZAN_2_PID_DATA"	// DB 231
AUTHOR : SIMATIC
FAMILY : CONTROL
VERSION : 0.0
"TCONT_CP"
BEGIN
END_DATA_BLOCK

DATA_BLOCK DB 232
VERSION : 0.0
"TEST_BLOGU"
BEGIN
END_DATA_BLOCK

ORGANIZATION_BLOCK OB 1
VERSION : 0.1
VAR_TEMP
  TEMP0 : BYTE ;
  TEMP1 : BYTE ;
  TEMP2 : BYTE ;
  TEMP3 : BYTE ;
  TEMP4 : BYTE ;
  TEMP5 : BYTE ;
  TEMP6 : INT ;
  TEMP7 : INT ;
  TEMP8 : INT ;
  TEMP9 : DATE_AND_TIME ;
END_VAR
BEGIN
NETWORK
TITLE =
      UC    "MAINBLOCK";
NETWORK
TITLE =
      CALL  "SCALE" (
           $1                       := P#P 292.0,
           $2                       := L#1092616192,
           $3                       := L#0,
           $4                       := "ALWAYS OFF",
           $5                       := "AI-SENSOR-DATA".HAT_BASINCI_RET_V,
           $6                       := "AI-SENSOR-DATA".HAT_BASINCI_ANLIK);
      CALL  "SCALE" (
           $1                       := P#P 294.0,
           $2                       := L#1092616192,
           $3                       := L#0,
           $4                       := "ALWAYS OFF",
           $5                       := "AI-SENSOR-DATA".HAVA_BASINCI_RET_V,
           $6                       := "AI-SENSOR-DATA".HAVA_BASINCI_ANLIK);
NETWORK
TITLE =
END_ORGANIZATION_BLOCK

ORGANIZATION_BLOCK "PID BLOCK"	// OB 35
VERSION : 0.1
VAR_TEMP
  TEMP0 : BYTE ;
  TEMP1 : BYTE ;
  TEMP2 : BYTE ;
  TEMP3 : BYTE ;
  TEMP4 : BYTE ;
  TEMP5 : BYTE ;
  TEMP6 : WORD ;
  TEMP7 : INT ;
  TEMP8 : INT ;
  TEMP9 : DATE_AND_TIME ;
END_VAR
BEGIN
NETWORK
TITLE =
      CALL  "JEN1_PID_KONTROL" , DB 52;
      CALL  "JEN2_PID_KONTROL" , "JEN2_KONTROL_BLOGU_DB";
NETWORK
TITLE =
      CALL  "KAZAN_1_PID_KONTROL" , DB 131;
      CALL  "KAZAN_2_PID_KONTROL" , DB 132;
END_ORGANIZATION_BLOCK

ORGANIZATION_BLOCK "ZAMANHATASI"	// OB 80
VERSION : 0.1
VAR_TEMP
  TEMP0 : BYTE ;
  TEMP1 : BYTE ;
  TEMP2 : BYTE ;
  TEMP3 : BYTE ;
  TEMP4 : BYTE ;
  TEMP5 : BYTE ;
  TEMP6 : WORD ;
  TEMP7 : BYTE ;
  TEMP8 : BYTE ;
  TEMP9 : BYTE ;
  TEMP10 : BYTE ;
  TEMP11 : DATE_AND_TIME ;
END_VAR
BEGIN
NETWORK
TITLE =
END_ORGANIZATION_BLOCK

ORGANIZATION_BLOCK "GERILIMHATASI"	// OB 81
VERSION : 0.1
VAR_TEMP
  TEMP0 : BYTE ;
  TEMP1 : BYTE ;
  TEMP2 : BYTE ;
  TEMP3 : BYTE ;
  TEMP4 : BYTE ;
  TEMP5 : BYTE ;
  TEMP6 : WORD ;
  TEMP7 : BYTE ;
  TEMP8 : BYTE ;
  TEMP9 : BYTE ;
  TEMP10 : BYTE ;
  TEMP11 : DATE_AND_TIME ;
END_VAR
BEGIN
NETWORK
TITLE =
END_ORGANIZATION_BLOCK

ORGANIZATION_BLOCK "HATAUYARISI"	// OB 82
VERSION : 0.1
VAR_TEMP
  TEMP0 : BYTE ;
  TEMP1 : BYTE ;
  TEMP2 : BYTE ;
  TEMP3 : BYTE ;
  TEMP4 : BYTE ;
  TEMP5 : BYTE ;
  TEMP6 : WORD ;
  TEMP7 : BOOL ;
  TEMP8 : BOOL ;
  TEMP9 : BOOL ;
  TEMP10 : BOOL ;
  TEMP11 : BOOL ;
  TEMP12 : BOOL ;
  TEMP13 : BOOL ;
  TEMP14 : BOOL ;
  TEMP15 : BYTE ;
  TEMP16 : BOOL ;
  TEMP17 : BOOL ;
  TEMP18 : BOOL ;
  TEMP19 : BOOL ;
  TEMP20 : BOOL ;
  TEMP21 : BOOL ;
  TEMP22 : BOOL ;
  TEMP23 : BOOL ;
  TEMP24 : BOOL ;
  TEMP25 : BOOL ;
  TEMP26 : BOOL ;
  TEMP27 : BOOL ;
  TEMP28 : BOOL ;
  TEMP29 : BOOL ;
  TEMP30 : BOOL ;
  TEMP31 : BOOL ;
  TEMP32 : DATE_AND_TIME ;
END_VAR
BEGIN
NETWORK
TITLE =
END_ORGANIZATION_BLOCK

ORGANIZATION_BLOCK "TAKMACIKARMAHATASI"	// OB 83
VERSION : 0.1
VAR_TEMP
  TEMP0 : BYTE ;
  TEMP1 : BYTE ;
  TEMP2 : BYTE ;
  TEMP3 : BYTE ;
  TEMP4 : BYTE ;
  TEMP5 : BYTE ;
  TEMP6 : WORD ;
  TEMP7 : INT ;
  TEMP8 : WORD ;
  TEMP9 : DATE_AND_TIME ;
END_VAR
BEGIN
NETWORK
TITLE =
END_ORGANIZATION_BLOCK

ORGANIZATION_BLOCK "CPUHARDWAREERROR"	// OB 84
VERSION : 0.1
VAR_TEMP
  TEMP0 : BYTE ;
  TEMP1 : BYTE ;
  TEMP2 : BYTE ;
  TEMP3 : BYTE ;
  TEMP4 : BYTE ;
  TEMP5 : BYTE ;
  TEMP6 : WORD ;
  TEMP7 : DWORD ;
  TEMP8 : DATE_AND_TIME ;
END_VAR
BEGIN
NETWORK
TITLE =
END_ORGANIZATION_BLOCK

ORGANIZATION_BLOCK "PROGRAMHATASI"	// OB 85
VERSION : 0.1
VAR_TEMP
  TEMP0 : BYTE ;
  TEMP1 : BYTE ;
  TEMP2 : BYTE ;
  TEMP3 : BYTE ;
  TEMP4 : BYTE ;
  TEMP5 : BYTE ;
  TEMP6 : INT ;
  TEMP7 : BYTE ;
  TEMP8 : BYTE ;
  TEMP9 : BYTE ;
  TEMP10 : BYTE ;
  TEMP11 : DATE_AND_TIME ;
END_VAR
BEGIN
NETWORK
TITLE =
END_ORGANIZATION_BLOCK

ORGANIZATION_BLOCK "RACKHATASI"	// OB 86
VERSION : 0.1
VAR_TEMP
  TEMP0 : BYTE ;
  TEMP1 : BYTE ;
  TEMP2 : BYTE ;
  TEMP3 : BYTE ;
  TEMP4 : BYTE ;
  TEMP5 : BYTE ;
  TEMP6 : WORD ;
  TEMP7 : ARRAY  [0 .. 31 ] OF BOOL ;
  TEMP8 : DATE_AND_TIME ;
END_VAR
BEGIN
NETWORK
TITLE =
END_ORGANIZATION_BLOCK

ORGANIZATION_BLOCK "HABERLESMEHATASI"	// OB 87
VERSION : 0.1
VAR_TEMP
  TEMP0 : BYTE ;
  TEMP1 : BYTE ;
  TEMP2 : BYTE ;
  TEMP3 : BYTE ;
  TEMP4 : BYTE ;
  TEMP5 : BYTE ;
  TEMP6 : WORD ;
  TEMP7 : DWORD ;
  TEMP8 : DATE_AND_TIME ;
END_VAR
BEGIN
NETWORK
TITLE =
END_ORGANIZATION_BLOCK

ORGANIZATION_BLOCK "COMPLETE RESTART"	// OB 100
VERSION : 0.1
VAR_TEMP
  TEMP0 : BYTE ;
  TEMP1 : BYTE ;
  TEMP2 : BYTE ;
  TEMP3 : BYTE ;
  TEMP4 : BYTE ;
  TEMP5 : BYTE ;
  TEMP6 : WORD ;
  TEMP7 : DWORD ;
  TEMP8 : DATE_AND_TIME ;
END_VAR
BEGIN
NETWORK
TITLE =
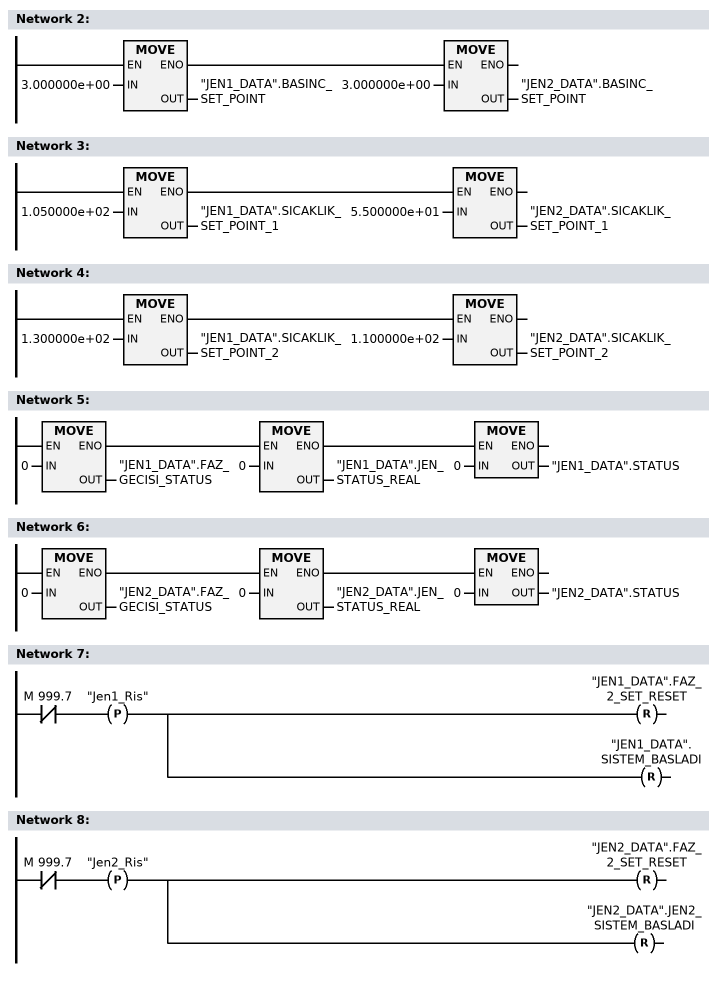
NETWORK
TITLE =
      A(;
      L     3.000000e+00;
      T     "JEN1_DATA".BASINC_SET_POINT;
      SET;
      SAVE;
      CLR;
      A     BR;
      );
      JNB   _001;
      L     3.000000e+00;
      T     "JEN2_DATA".BASINC_SET_POINT;
_001: NOP   0;
NETWORK
TITLE =
      A(;
      L     1.050000e+02;
      T     "JEN1_DATA".SICAKLIK_SET_POINT_1;
      SET;
      SAVE;
      CLR;
      A     BR;
      );
      JNB   _002;
      L     5.500000e+01;
      T     "JEN2_DATA".SICAKLIK_SET_POINT_1;
_002: NOP   0;
NETWORK
TITLE =
      A(;
      L     1.300000e+02;
      T     "JEN1_DATA".SICAKLIK_SET_POINT_2;
      SET;
      SAVE;
      CLR;
      A     BR;
      );
      JNB   _003;
      L     1.100000e+02;
      T     "JEN2_DATA".SICAKLIK_SET_POINT_2;
_003: NOP   0;
NETWORK
TITLE =
      A(;
      A(;
      L     0;
      T     "JEN1_DATA".FAZ_GECISI_STATUS;
      SET;
      SAVE;
      CLR;
      A     BR;
      );
      JNB   _004;
      L     0;
      T     "JEN1_DATA".JEN_STATUS_REAL;
      SET;
      SAVE;
      CLR;
_004: A     BR;
      );
      JNB   _005;
      L     0;
      T     "JEN1_DATA".STATUS;
_005: NOP   0;
NETWORK
TITLE =
      A(;
      A(;
      L     0;
      T     "JEN2_DATA".FAZ_GECISI_STATUS;
      SET;
      SAVE;
      CLR;
      A     BR;
      );
      JNB   _006;
      L     0;
      T     "JEN2_DATA".JEN_STATUS_REAL;
      SET;
      SAVE;
      CLR;
_006: A     BR;
      );
      JNB   _007;
      L     0;
      T     "JEN2_DATA".STATUS;
_007: NOP   0;
NETWORK
TITLE =
      AN    M 999.7;
      FP    "Jen1_Ris";
      R     "JEN1_DATA".FAZ_2_SET_RESET;
      R     "JEN1_DATA".SISTEM_BASLADI;
NETWORK
TITLE =
      AN    M 999.7;
      FP    "Jen2_Ris";
      R     "JEN2_DATA".FAZ_2_SET_RESET;
      R     "JEN2_DATA".JEN2_SISTEM_BASLADI;
END_ORGANIZATION_BLOCK

ORGANIZATION_BLOCK "RESTART"	// OB 101
VERSION : 0.1
VAR_TEMP
  TEMP0 : BYTE ;
  TEMP1 : BYTE ;
  TEMP2 : BYTE ;
  TEMP3 : BYTE ;
  TEMP4 : BYTE ;
  TEMP5 : BYTE ;
  TEMP6 : WORD ;
  TEMP7 : DWORD ;
  TEMP8 : DATE_AND_TIME ;
END_VAR
BEGIN
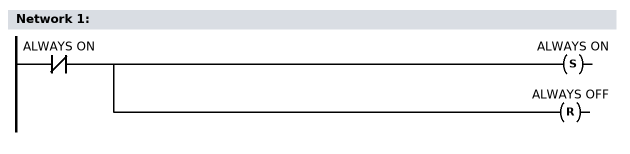
NETWORK
TITLE =
      AN    "ALWAYS ON";
      S     "ALWAYS ON";
      R     "ALWAYS OFF";
END_ORGANIZATION_BLOCK

ORGANIZATION_BLOCK "COLD RESTART"	// OB 102
VERSION : 0.1
VAR_TEMP
  TEMP0 : BYTE ;
  TEMP1 : BYTE ;
  TEMP2 : BYTE ;
  TEMP3 : BYTE ;
  TEMP4 : BYTE ;
  TEMP5 : BYTE ;
  TEMP6 : WORD ;
  TEMP7 : DWORD ;
  TEMP8 : DATE_AND_TIME ;
END_VAR
BEGIN
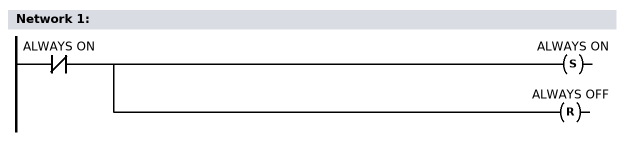
NETWORK
TITLE =
      AN    "ALWAYS ON";
      S     "ALWAYS ON";
      R     "ALWAYS OFF";
END_ORGANIZATION_BLOCK

ORGANIZATION_BLOCK "PROGRAMMINGERROR"	// OB 121
VERSION : 0.1
VAR_TEMP
  TEMP0 : BYTE ;
  TEMP1 : BYTE ;
  TEMP2 : BYTE ;
  TEMP3 : BYTE ;
  TEMP4 : BYTE ;
  TEMP5 : BYTE ;
  TEMP6 : WORD ;
  TEMP7 : WORD ;
  TEMP8 : WORD ;
  TEMP9 : DATE_AND_TIME ;
END_VAR
BEGIN
NETWORK
TITLE =
END_ORGANIZATION_BLOCK

ORGANIZATION_BLOCK "MOD_ERR"	// OB 122
TITLE = "Module Access Error"
VERSION : 0.1
VAR_TEMP
  OB122_EV_CLASS : BYTE ;	//16#29, Event class 2, Entering event state, Internal fault event
  OB122_SW_FLT : BYTE ;	//16#XX Software error code
  OB122_PRIORITY : BYTE ;	//Priority of OB Execution
  OB122_OB_NUMBR : BYTE ;	//122 (Organization block 122, OB122)
  OB122_BLK_TYPE : BYTE ;	//16#88/8C/8E Type of block fault occured in
  OB122_MEM_AREA : BYTE ;	//Memory area where access error occured
  OB122_MEM_ADDR : WORD ;	//Memory address where access error occured
  OB122_BLK_NUM : WORD ;	//Block number in which error occured
  OB122_PRG_ADDR : WORD ;	//Program address where error occured
  OB122_DATE_TIME : DATE_AND_TIME ;	//Date and time OB1 started
END_VAR
BEGIN
// (block stored without names or comments; labels and parameter names are numbered)
END_ORGANIZATION_BLOCK

DATA_BLOCK DB 100
VERSION : 0.1
  STRUCT
   JEN1_Min_Basinc : REAL  := 5.000000e+000;	//Jenerator 1 min otomatik sekans basinci
   JEN1_Max_Basinc : REAL  := 5.500000e+000;	//Jenerator 1 max otomatik sekans basinci
   JEN2_Min_Basinc : REAL  := 5.000000e+000;	//Jenerator 2 min otomatik sekans basinci
   JEN2_Max_Basinc : REAL  := 5.500000e+000;	//Jenerator 2 max otomatik sekans basinci
   OTOKLAV_First_Oran : REAL  := 2.000000e+001;	//Otoklav oransal vana otomatik sekans ilk acilis orani
   OTOKLAV_Kademeli_Artis : REAL  := 5.000000e+000;	//Otoklav oransal vana kademeli artis katsayisi
   Otoklav_1_TimeData : STRUCT 	//Otoklav 1 hmi süre bilgisi
    Hours : INT ;	//Istenen calisma saati
    Minutes : INT  := 30;	//Istenen calisma dakikasi
    Second : INT ;	//Istenen calisma saniyesi
   END_STRUCT ;
   Otoklav_2_TimeData : STRUCT 	//Otoklav 2 hmi süre bilgisi
    Hours : INT ;	//Istenen calisma saati
    Minutes : INT  := 30;	//Istenen calisma dakikasi
    Second : INT ;	//Istenen calisma saniyesi
   END_STRUCT ;
   O_VanaAciklikOrani : REAL  := 2.500000e+001;	//Oransal vana aciklik orani
   O_VanaKademeSayisi : REAL  := 5.000000e+000;	//Oransal vana kademeli artis katsayisi
   Otoklav1_Bos_Vanasi : STRUCT 	//Otoklav 1 Bosaltim Vanasi
    Vana_Acilma_Sayisi : INT  := 3;
    Periyod_Bekleme_Suresi : INT  := 120;	//Saniye bazinda
    Acik_Kalma_Suresi : INT  := 10;	//Saniye bazinda
   END_STRUCT ;
   Otoklav2_Bos_Vanasi : STRUCT 	//Otoklav 2 Bosaltim Vanasi
    Vana_Acilma_Sayisi : INT  := 3;
    Periyod_Bekleme_Suresi : INT  := 120;	//Saniye bazinda
    Acik_Kalma_Suresi : INT  := 10;	//Saniye bazinda
   END_STRUCT ;
  END_STRUCT ;	
BEGIN
   JEN1_Min_Basinc := 5.000000e+00;
   JEN1_Max_Basinc := 5.500000e+00;
   JEN2_Min_Basinc := 5.000000e+00;
   JEN2_Max_Basinc := 5.500000e+00;
   Otoklav_1_TimeData.Minutes := 21;
   Otoklav_2_TimeData.Minutes := 21;
   O_VanaAciklikOrani := 3.000000e+01;
   O_VanaKademeSayisi := 5.000000e+00;
   Otoklav1_Bos_Vanasi.Vana_Acilma_Sayisi := 5;
   Otoklav1_Bos_Vanasi.Periyod_Bekleme_Suresi := 60;
   Otoklav1_Bos_Vanasi.Acik_Kalma_Suresi := 7;
   Otoklav2_Bos_Vanasi.Vana_Acilma_Sayisi := 5;
   Otoklav2_Bos_Vanasi.Periyod_Bekleme_Suresi := 60;
   Otoklav2_Bos_Vanasi.Acik_Kalma_Suresi := 7;
END_DATA_BLOCK

ORGANIZATION_BLOCK OB 1
TITLE = "Main Program Sweep (Cycle)"
VERSION : 0.1
VAR_TEMP
  OB1_EV_CLASS : BYTE ;	//Bits 0-3 = 1 (Coming event), Bits 4-7 = 1 (Event class 1)
  OB1_SCAN_1 : BYTE ;	//1 (Cold restart scan 1 of OB 1), 3 (Scan 2-n of OB 1)
  OB1_PRIORITY : BYTE ;	//Priority of OB Execution
  OB1_OB_NUMBR : BYTE ;	//1 (Organization block 1, OB1)
  OB1_RESERVED_1 : BYTE ;	//Reserved for system
  OB1_RESERVED_2 : BYTE ;	//Reserved for system
  OB1_PREV_CYCLE : INT ;	//Cycle time of previous OB1 scan (milliseconds)
  OB1_MIN_CYCLE : INT ;	//Minimum cycle time of OB1 (milliseconds)
  OB1_MAX_CYCLE : INT ;	//Maximum cycle time of OB1 (milliseconds)
  OB1_DATE_TIME : DATE_AND_TIME ;	//Date and time OB1 started
END_VAR
BEGIN
// (block stored without names or comments; labels and parameter names are numbered)
END_ORGANIZATION_BLOCK
